// TwinCAT 3 PLC project Sample02
// ProgramVersion: 3.1.4020.1
// libraries:
//   Tc2_Standard, * (Beckhoff Automation GmbH)
//   Tc2_System, * (Beckhoff Automation GmbH)
//   Tc3_Module, * (Beckhoff Automation GmbH)
// project tree:
//   / PlcTask.TcTTO
//   POUs/ F_CalcSum1DimArray.TcPOU, MAIN.TcPOU
// real-time tasks:
//   TASK PlcTask: cycle T#10ms, priority 20, ADS port 350

CONFIGURATION Sample02
    RESOURCE PLC ON TwinCAT3
        TASK PlcTask(INTERVAL := T#10ms, PRIORITY := 20);
        PROGRAM MAIN WITH PlcTask : MAIN;
    END_RESOURCE
END_CONFIGURATION

// ---- POUs/MAIN.TcPOU
PROGRAM MAIN
VAR
	array01 		: ARRAY[2..8] OF LREAL := [16.1, 34.1, 4.1, 43.1, 35.1, 2.1, 65.1];
	lrSum01			: LREAL;
	
	array02 		: ARRAY[-1..2] OF LREAL := [16.1, 34.1, 9.1, 13.1];
	lrSum02			: LREAL;
	
	array03 		: ARRAY[-3..-1] OF LREAL := [16.1, 34.1, 8.1];
	lrSum03			: LREAL;
END_VAR

lrSum01 := F_CalcSum1DimArray(array01);
lrSum02 := F_CalcSum1DimArray(array02);
lrSum03 := F_CalcSum1DimArray(array03);

END_PROGRAM

// ---- POUs/F_CalcSum1DimArray.TcPOU
FUNCTION F_CalcSum1DimArray : LREAL
VAR_IN_OUT
	arrData		: ARRAY[*] OF LREAL;
END_VAR
VAR
	nIndex		: DINT;
END_VAR

F_CalcSum1DimArray := 0;
FOR nIndex := LOWER_BOUND(arrData, 1) TO UPPER_BOUND(arrData, 1) DO
	F_CalcSum1DimArray := F_CalcSum1DimArray + arrData[nIndex];
END_FOR

END_FUNCTION
